# EPICS IOC start-up script: iocsh/AH501.iocsh
# ### AH501.iocsh ###

#- ###################################################
#- PREFIX         - IOC Prefix
#- INSTANCE       - Name of quadEM port instance to create
#- IP_ADDR        - IP address of AH501
#- QUADEM         - Location of quadEM module
#- ASYN           - Location of asyn module
#- MODEL          - Optional: AH501 Model (AH501/AH501C/AH501D)
#-                  Default: AH501
#-
#- RING_SIZE      - Optional: Ring Size
#-                  Default: 10000
#- ###################################################

drvAsynIPPortConfigure("IP_$(INSTANCE)", "$(IP_ADDR)", 0, 0, 0)
asynOctetSetInputEos("IP_$(INSTANCE)",  0, "\r\n")
asynOctetSetOutputEos("IP_$(INSTANCE)", 0, "\r")

dbLoadRecords("$(ASYN)/db/asynRecord.db", "P=$(PREFIX), R=asyn_IP_$(INSTANCE),PORT=IP_$(INSTANCE),ADDR=0,OMAX=256,IMAX=256")

drvAHxxxConfigure("$(INSTANCE)", "IP_$(INSTANCE)", $(RING_SIZE=10000), "$(MODEL=AH501)")

dbLoadRecords("$(QUADEM)/db/AH501.template", "P=$(PREFIX), R=$(INSTANCE):, PORT=$(INSTANCE)")
